FUNCTION_BLOCK FB_Toggle
VAR_INPUT
	Timer : TIME;
END_VAR
VAR_OUTPUT
	Toggle_Out : BOOL;
END_VAR
VAR
	Timer_Out : BOOL;
	Timer_Toggle: TON;
END_VAR

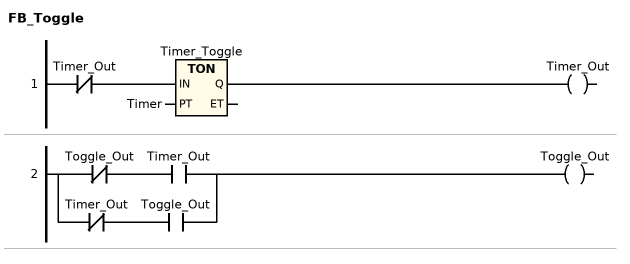
// NETWORK 1
Timer_Toggle(IN := NOT Timer_Out, PT := Timer); // TON
Timer_Out := Timer_Toggle.Q;

// NETWORK 2
Toggle_Out := NOT Toggle_Out AND Timer_Out OR NOT Timer_Out AND Toggle_Out;

END_FUNCTION_BLOCK

(* stored: Version 1.1.0.1, ProductVersion 3.1.4024.6
   POU FB_Toggle: Id {3014dbb5-bccc-4063-8ec9-b8cdb297ccae}, SpecialFunc None *)
